{attribute 'pack_mode' := '1'}
TYPE ST_HomeAxis EXTENDS ST_MsgToPLC:
STRUCT
    axisIndex: DINT;
END_STRUCT
END_TYPE

(* stored: Version 1.1.0.1, ProductVersion 3.1.4022.18
   DUT ST_HomeAxis: Id {06aead2c-fc92-4f56-9b66-cf2ac1527113} *)
